FUNCTION "SM_Changed" : Bool
{ S7_Optimized_Access := 'FALSE' }
VERSION : 0.1
   VAR_IN_OUT
      inst : "typeSM";
   END_VAR


BEGIN
	#SM_Changed := #inst.stateChanged;
END_FUNCTION

